// TwinCAT 3 PLC project Oefeningen3
// ProgramVersion: 3.1.4026.18
// libraries:
//   Tc2_Standard, * (Beckhoff Automation GmbH)
//   Tc2_System, * (Beckhoff Automation GmbH)
//   Tc3_Module, * (Beckhoff Automation GmbH)
// project tree:
//   / GlobalTextList.TcGTLO, PlcTask.TcTTO, Visualization Manager.TcVMO (not stored)
//   POUs/ MAIN.TcPOU, prg_AutomatischeDeur.TcPOU, prg_Belsignaal.TcPOU, prg_DraaiRichtingMotor.TcPOU, prg_Knipperlicht.TcPOU, prg_Millis.TcPOU, prg_OpenbaarToilet.TcPOU, prg_Parking.TcPOU, prg_ProductenTellen.TcPOU, prg_Setpointsturing.TcPOU, prg_Startveiligheid.TcPOU, prg_Teleruptor.TcPOU, prg_TrappenhuisautomaatTijdsinstelling.TcPOU, prg_TrappenhuisautomaatVerlenging.TcPOU
//   VISUs/ Visualization_SetPoint.TcVIS
// (motion and I/O tree: see PLC project oefeningen1)
// real-time tasks:
//   TASK PlcTask: cycle T#10ms, priority 20, ADS port 350
//   TASK PlcTask1: cycle T#10ms, priority 21, ADS port 351
//   TASK PlcTask2: cycle T#10ms, priority 22, ADS port 352
//   TASK PlcTask3: cycle T#10ms, priority 23, ADS port 353
//   TASK PlcTask4: cycle T#10ms, priority 24, ADS port 354

CONFIGURATION Oefeningen3
    RESOURCE PLC ON TwinCAT3
        TASK PlcTask(INTERVAL := T#10ms, PRIORITY := 22);
        PROGRAM MAIN WITH PlcTask : MAIN;
    END_RESOURCE
END_CONFIGURATION

// ---- POUs/MAIN.TcPOU
PROGRAM MAIN
VAR
END_VAR

//prg_Teleruptor();
//prg_Startveiligheid();
//prg_TrappenhuisautomaatVerlenging();
//prg_TrappenhuisautomaatTijdsinstelling();
//prg_Knipperlicht();
//prg_Millis();
//prg_OpenbaarToilet();
//prg_AutomatischeDeur();
//prg_Setpointsturing();
//prg_DraaiRichtingMotor();
//prg_Belsignaal();
//prg_Parking();
//prg_ProductenTellen();

END_PROGRAM

// ---- POUs/prg_AutomatischeDeur.TcPOU
PROGRAM prg_AutomatischeDeur
VAR
	bHoofdSchakelaar		AT		%I*			:BOOL;
	bDrukknop				AT		%I*			:BOOL;
	bSensor					AT		%I*			:BOOL;
	
	bDeur					AT		%Q*			:BOOL;
	DeurDicht: TOF;
END_VAR

DeurDicht(IN:= bHoofdSchakelaar AND (bDrukknop OR bSensor), PT:= T#1S, Q=> bDeur);

END_PROGRAM

// ---- POUs/prg_Belsignaal.TcPOU
PROGRAM prg_Belsignaal
VAR
	Sensor1, Sensor2		AT		%I*		:BOOL;
	Bel						AT		%Q*		:BOOL;
	bBinnen          : BOOL;
	BinnenKomen: R_TRIG;
	BuitenGaan: R_TRIG;
END_VAR

BinnenKomen(CLK := Sensor1);
BuitenGaan(CLK := Sensor2);

IF BinnenKomen.Q AND NOT Sensor2 THEN
    bBinnen := TRUE;      // S01 eerst → binnen
ELSIF BuitenGaan.Q AND NOT Sensor1 THEN
    bBinnen := FALSE;     // S02 eerst → buiten
END_IF

Bel := bBinnen AND (Sensor1 OR Sensor2);

END_PROGRAM

// ---- POUs/prg_DraaiRichtingMotor.TcPOU
PROGRAM prg_DraaiRichtingMotor
VAR
	bSensorA	AT		%I*		:BOOL;
	bSensorB	AT		%I*		:BOOL;
	
	bLinks		AT		%Q*		:BOOL;
	bRechts		AT		%Q*		:BOOL;
	bMotor		AT		%Q*		:BOOL;
	bAlarm		AT		%Q*		:BOOL;
	Links: R_TRIG;
	Rechts: R_TRIG;
END_VAR

Links(CLK:= bSensorA, Q=> bLinks);
Rechts(CLK:= bSensorB, Q=> bRechts);

IF bLinks THEN
	bMotor:=TRUE;
	bAlarm:=FALSE;
ELSIF bRechts THEN
	bMotor:=FALSE;
	bAlarm:=TRUE;
END_IF

END_PROGRAM

// ---- POUs/prg_Knipperlicht.TcPOU
PROGRAM prg_Knipperlicht
VAR
	bLamp				AT		%Q*		:BOOL;
	TimerOn: TON;
	TimerOff: TOF;
	
	//UitBreiding:
	nPotentioMeter		AT		%I*		:INT;
	Knipperfrequentie	:REAL;
	bLamp1				AT		%Q*		:BOOL;
	bLamp2				AT		%Q*		:BOOL;
	SpanningPot			AT		%Q*		:REAL;
END_VAR

//TimerOn(IN:= NOT(bLamp), PT:= T#500MS);
//TimerOff(IN:= TimerOn.Q, PT:= T#500MS, Q=> bLamp);

//Uitbreiding:
SpanningPot:= INT_TO_REAL(nPotentioMeter) * 10 / 32767;

IF (SpanningPot < 2) THEN //Frequentie 0.5Hz = 1s aan, 1s Uit
TimerOn(IN:= NOT(bLamp1), PT:= T#1S);
TimerOff(IN:= TimerOn.Q, PT:= T#1S, Q=> bLamp1);
bLamp2 := FALSE;
	ELSIF (SpanningPot >= 2) AND (SpanningPot < 4) THEN //1 Hz (500ms ON / 500ms OFF)
	TimerOn(IN:= NOT(bLamp1), PT:= T#500MS);
	TimerOff(IN:= TimerOn.Q, PT:= T#500MS, Q=> bLamp1);
	bLamp2 := FALSE;
		ELSIF (SpanningPot >= 4) AND (SpanningPot < 6) THEN //2 Hz (250ms ON / 250ms OFF)
		TimerOn(IN:= NOT(bLamp1), PT:= T#250MS);
		TimerOff(IN:= TimerOn.Q, PT:= T#250MS, Q=> bLamp1);
		bLamp2 := FALSE;
			ELSIF (SpanningPot >= 6) THEN //5Hz => 1000ms / 5 = 200ms => 200ms / 2 = 100ms AAN, 100ms UIT
			TimerOn(IN:= NOT(bLamp1), PT:= T#100MS);
			TimerOff(IN:= TimerOn.Q, PT:= T#100MS, Q=> bLamp1);
			bLamp2 := NOT(bLamp1);
END_IF

END_PROGRAM

// ---- POUs/prg_Millis.TcPOU
PROGRAM prg_Millis
VAR
	tpMillis : TP;
	bPuls	AT		%Q*		:BOOL;
END_VAR

tpMillis(IN := NOT tpMillis.Q, PT := T#1S);
bPuls := NOT(tpMillis.Q);

//Als je dit in 1 regel wilt moet je gewoon bPuls bij de Q van tpmillis zetten

END_PROGRAM

// ---- POUs/prg_OpenbaarToilet.TcPOU
PROGRAM prg_OpenbaarToilet
VAR
	bSchakel1, bSchakel2, bSchakel3		AT		%I*		:BOOL;
	bLamp1, bLamp2, bLamp3				AT		%Q*		:BOOL;
	bVentilator							AT		%Q*		:BOOL;
	TimerOff: TOF;
END_VAR

bLamp1:= bSchakel1;
bLamp2:= bSchakel2;
bLamp3:= bSchakel3;
TimerOff(IN:= bSchakel1 OR bSchakel2 OR bSchakel3, PT:= T#5S, Q=> bVentilator);
//Dit werkt omdat de TOF op de FALLING EDGE detecteerd

END_PROGRAM

// ---- POUs/prg_Parking.TcPOU
PROGRAM prg_Parking
VAR
	Sensor1, Sensor2    AT	 	%I*		:BOOL;
	bBinnen               : BOOL;
 	Slagboom       		AT 		%Q* 	:BOOL;
	Roodlicht			AT		%Q*		:BOOL;
	Groenlicht			AT		%Q*		:BOOL;
	AantalAutos			AT		%Q*		:INT;
	AutoTeller: CTUD;
	BinnenRising: R_TRIG;
	BuitenRising: R_TRIG;
	BinnenFalling: F_TRIG;
	BuitenFalling: F_TRIG;
END_VAR

BinnenRising(CLK := Sensor1);
BuitenRising(CLK := Sensor2);
BinnenFalling(CLK := Sensor1);
BuitenFalling(CLK := Sensor2);

(* Richting bepalen *)
IF BinnenRising.Q AND NOT Sensor2 THEN
	bBinnen := TRUE;          // binnenrijden
ELSIF BuitenRising.Q AND NOT Sensor1 THEN
	bBinnen := FALSE;         // buitengaan
END_IF

(* Slagboom *)
Slagboom := (Sensor1 OR Sensor2)
            AND (NOT bBinnen OR (AutoTeller.CV < AutoTeller.PV));

(* Teller *)
AutoTeller(
	CU := (bBinnen AND BuitenFalling.Q),
	CD := (NOT bBinnen AND BinnenFalling.Q),
	LOAD := FALSE,
	PV := 10
);

(* Verkeerslichten *)
IF AutoTeller.CV >= AutoTeller.PV THEN
	Roodlicht := TRUE;
	Groenlicht := FALSE;
ELSE
	Groenlicht := TRUE;
	Roodlicht := FALSE;
END_IF

(* Visualisatie tellerstand *)
AantalAutos := AutoTeller.CV * 32767 / 10;

END_PROGRAM

// ---- POUs/prg_ProductenTellen.TcPOU
PROGRAM prg_ProductenTellen
VAR
	bSensor		AT		%I*		:BOOL;
	
	bKlep		AT		%Q*		:BOOL; //0 is rechtdoor, 1 is afgebogen
	CounterRechtdoor: CTU;
	CounterAfslaan: CTU;
END_VAR

IF 	NOT(bKlep) THEN
CounterRechtdoor(
	CU:= bSensor, 
	PV:= 10);
END_IF

IF CounterRechtdoor.Q THEN
	bKlep := 1;
	CounterRechtdoor.RESET := TRUE;
END_IF

IF bKlep THEN
CounterAfslaan(
	CU:= bSensor,  
	PV:= 20,);
END_IF

IF CounterAfslaan.Q THEN
	bKlep := 0;
	CounterAfslaan.RESET := TRUE;
END_IF

END_PROGRAM

// ---- POUs/prg_Setpointsturing.TcPOU
PROGRAM prg_Setpointsturing
VAR
	DrukPlus, DrukMin		AT		%I*		:BOOL;
	SetPoint		:INT:=0;
	LangerAls1sec: TON;
	LANGEPLUS: TON;
	LANGEMIN: TON;
	FallingDrukPlus: F_TRIG;
	FallingDrukMin: F_TRIG;
	SpanningUit		AT			%Q*			:REAL;
END_VAR

LANGEPLUS(IN := DrukPlus, PT := T#1S);
LANGEMIN(IN := DrukMin,  PT := T#1S);

LangerAls1sec(IN := LANGEPLUS.Q OR LANGEMIN.Q, PT := T#1S);

FallingDrukPlus(CLK := DrukPlus);
FallingDrukMin(CLK := DrukMin);

(* Lange druk: 100 per seconde *)
IF LangerAls1sec.Q THEN
    IF LANGEPLUS.Q THEN
        SetPoint := SetPoint + 100;
    ELSIF LANGEMIN.Q THEN
        SetPoint := SetPoint - 100;
    END_IF
    LangerAls1sec(IN := FALSE);   (* timer herstarten *)
END_IF

(* Korte druk *)
IF FallingDrukPlus.Q AND NOT LANGEPLUS.Q THEN
    SetPoint := SetPoint + 1;
ELSIF FallingDrukMin.Q AND NOT LANGEMIN.Q THEN
    SetPoint := SetPoint - 1;
END_IF

(* Begrenzing *)
IF SetPoint > 1000 THEN SetPoint := 1000; END_IF
IF SetPoint < 0 THEN SetPoint := 0; END_IF

SpanningUit := INT_TO_REAL(SetPoint) * 10.0 / 1000.0;

END_PROGRAM

// ---- POUs/prg_Startveiligheid.TcPOU
PROGRAM prg_Startveiligheid
VAR
	bStart			AT		%I*		:BOOL;
	
	bMachine		AT		%Q*		:BOOL;
	fbStart: TON;
END_VAR

fbStart(IN:= bStart, PT:= T#5S, Q=> bMachine);

END_PROGRAM

// ---- POUs/prg_Teleruptor.TcPOU
PROGRAM prg_Teleruptor
VAR
	bDruk1Keuken, bDruk2Living, bDruk3Gang		AT		%I*		:BOOL;
	
	bKeuken		AT		%Q*		:BOOL;
	fbKeuken: TP;
END_VAR

fbKeuken(IN:= bDruk1Keuken OR bDruk2Living OR bDruk3Gang, PT:= T#10s, Q=> bKeuken);

END_PROGRAM

// ---- POUs/prg_TrappenhuisautomaatTijdsinstelling.TcPOU
PROGRAM prg_TrappenhuisautomaatTijdsinstelling
VAR
	bDrukknop1, bDrukknop2, bDrukknop3, bDrukknop4, bDrukknop5, bDrukknop6	AT	%I*	:BOOL;
	
	bVerlichting		AT		%Q*		:BOOL;

	fbVerlichting: TOF;
	RisingEdge: R_TRIG;
	bAanUit: BOOL;
END_VAR

RisingEdge(CLK:= bDrukknop1 OR bDrukknop2 OR bDrukknop3 OR bDrukknop4 OR bDrukknop5 OR bDrukknop6, Q=> bAanUit);

fbVerlichting(IN:= bAanUit, PT:= T#10S);
	
IF bAanUit AND bVerlichting THEN
	bVerlichting:=FALSE;
ELSIF bAanUit AND NOT bVerlichting THEN 
	bVerlichting:=fbVerlichting.Q;
END_IF

END_PROGRAM

// ---- POUs/prg_TrappenhuisautomaatVerlenging.TcPOU
PROGRAM prg_TrappenhuisautomaatVerlenging
VAR
	bDrukknop1, bDrukknop2, bDrukknop3, bDrukknop4, bDrukknop5, bDrukknop6	AT	%I*	:BOOL;
	
	bVerlichting		AT		%Q*		:BOOL;
	fbVerlichting: TOF;
END_VAR

fbVerlichting(IN:= bDrukknop1 OR bDrukknop2 OR bDrukknop3 OR bDrukknop4 OR bDrukknop5 OR bDrukknop6, PT:= T#3s, Q=> bVerlichting);

END_PROGRAM

// ---- GlobalTextList.TcGTLO
TEXTLIST GlobalTextList
  960 = 'DrukMin'
  500 = 'DrukPlus'
END_TEXTLIST

// ---- VISUs/Visualization_SetPoint.TcVIS
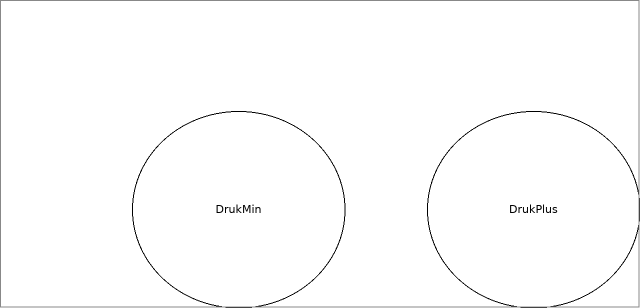
VISUALIZATION Visualization_SetPoint  // 640x308
    Ellipse (132,111 213x197), "DrukMin"
        tap prg_Setpointsturing.DrukMin
    Ellipse (427,111 213x197), "DrukPlus"
        tap prg_Setpointsturing.DrukPlus
END_VISUALIZATION
